// TwinCAT 3 PLC project SaftyPLC_1
// ProgramVersion: 3.1.4026.12
// libraries:
//   Tc2_Standard, * (Beckhoff Automation GmbH)
//   Tc2_System, * (Beckhoff Automation GmbH)
//   Tc2_Utilities, * (Beckhoff Automation GmbH)
//   Tc3_Module, * (Beckhoff Automation GmbH)
// project tree:
//   GVLs/ GVL_io.TcGVL, GVL_Safety.TcGVL
//   / PlcTask.TcTTO, XTS_Task.TcTTO (not stored)
//   POUs/ MAIN.TcPOU
// (motion and I/O tree: see PLC project planartrackmovement_1)
// real-time tasks:
//   TASK XTS Task: cycle T#500us, priority 1, ADS port 350
//   TASK Job Task: cycle default, priority 32
//   TASK MC-Task (MET): cycle T#2ms, priority 3, ADS port 521
//   TASK MC-Task (MPT): cycle T#10ms, priority 8, ADS port 531
//   TASK PlcTask: cycle T#1ms, priority 20, ADS port 351
//   TASK PlcTask1: cycle T#1ms, priority 21, ADS port 352
// variable links:
//   SaftyPLC_1/SaftyPLC_1 Instance <-> Device 1 (EtherCAT)/Term 1 (EK1200)/Term 13 (EL2912)
//     PlcTask Inputs/GVL_Safety.Error_Com <-> StandardInputs/TwinSafeGroup1.Error_Com_142
//     PlcTask Inputs/GVL_Safety.Error_Other <-> StandardInputs/TwinSafeGroup1.Error_Other_143
//     PlcTask Inputs/GVL_Safety.Error_Out <-> StandardInputs/TwinSafeGroup1.Error_out_141
//     PlcTask Inputs/GVL_Safety.SaeftyOk <-> StandardInputs/TwinSafeGroup1.SafetyOk_72
//     PlcTask Inputs/GVL_Safety.SafetyInRun <-> StandardInputs/TwinSafeGroup1.SafetyInRun_73
//     PlcTask Outputs/GVL_Safety.Reset <-> StandardOutputs/TwinSafeGroup1.ErrorAcknowledgement_1
//     PlcTask Outputs/GVL_Safety.Run <-> StandardOutputs/TwinSafeGroup1.Run_2
//     PlcTask Outputs/GVL_Safety.Start <-> StandardOutputs/TwinSafeGroup1.STO_75
//   SaftyPLC_1/SaftyPLC_1 Instance <-> Device 1 (EtherCAT)/Term 1 (EK1200)/Term 2 (EL1809)
//     PlcTask Inputs/GVL_Safety.HwReset <-> Channel 16/Input
//     PlcTask Inputs/GVL_Safety.HwStart <-> Channel 14/Input
//     PlcTask Inputs/GVL_Safety.HwStop <-> Channel 15/Input
//   SaftyPLC_1/SaftyPLC_1 Instance <-> Device 4 (EtherCAT)/Box 50 (AT5100-0100)
//     PlcTask Inputs/GVL_io.D_Spannung[5] <-> DRV Info data 1/D-Spannung
//     PlcTask Inputs/GVL_io.Q_Spannung[5] <-> DRV Info data 1/Q-Spannung
//     PlcTask Outputs/GVL_Safety.Reset <-> Module 1 (SAFETY)/SAFETY Standard Outputdata/Standard In Var 1
//     PlcTask Outputs/GVL_Safety.Run <-> Module 1 (SAFETY)/SAFETY Standard Outputdata/Standard In Var 5
//   SaftyPLC_1/SaftyPLC_1 Instance <-> Device 4 (EtherCAT)/Box 51 (AT5100-0100)
//     PlcTask Inputs/GVL_io.D_Spannung[6] <-> DRV Info data 1/D-Spannung
//     PlcTask Inputs/GVL_io.Q_Spannung[6] <-> DRV Info data 1/Q-Spannung
//     PlcTask Outputs/GVL_Safety.Reset <-> Module 1 (SAFETY)/SAFETY Standard Outputdata/Standard In Var 1
//     PlcTask Outputs/GVL_Safety.Run <-> Module 1 (SAFETY)/SAFETY Standard Outputdata/Standard In Var 5
//   SaftyPLC_1/SaftyPLC_1 Instance <-> Device 4 (EtherCAT)/Box 52 (AT5100-0100)
//     PlcTask Outputs/GVL_Safety.Reset <-> Module 1 (SAFETY)/SAFETY Standard Outputdata/Standard In Var 1
//     PlcTask Outputs/GVL_Safety.Run <-> Module 1 (SAFETY)/SAFETY Standard Outputdata/Standard In Var 5
//   SaftyPLC_1/SaftyPLC_1 Instance <-> Device 4 (EtherCAT)/Box 53 (AT5100-0100)
//     PlcTask Outputs/GVL_Safety.Reset <-> Module 1 (SAFETY)/SAFETY Standard Outputdata/Standard In Var 1
//     PlcTask Outputs/GVL_Safety.Run <-> Module 1 (SAFETY)/SAFETY Standard Outputdata/Standard In Var 5
//   SaftyPLC_1/SaftyPLC_1 Instance <-> Device 4 (EtherCAT)/Box 54 (AT5100-0100)
//     PlcTask Outputs/GVL_Safety.Reset <-> Module 1 (SAFETY)/SAFETY Standard Outputdata/Standard In Var 1
//     PlcTask Outputs/GVL_Safety.Run <-> Module 1 (SAFETY)/SAFETY Standard Outputdata/Standard In Var 5
//   SaftyPLC_1/SaftyPLC_1 Instance <-> Device 4 (EtherCAT)/Box 55 (AT5100-0100)
//     PlcTask Outputs/GVL_Safety.Reset <-> Module 1 (SAFETY)/SAFETY Standard Outputdata/Standard In Var 1
//     PlcTask Outputs/GVL_Safety.Run <-> Module 1 (SAFETY)/SAFETY Standard Outputdata/Standard In Var 5
//   SaftyPLC_1/SaftyPLC_1 Instance <-> Device 4 (EtherCAT)/Box 56 (AT5100-0100)
//     PlcTask Outputs/GVL_Safety.Reset <-> Module 1 (SAFETY)/SAFETY Standard Outputdata/Standard In Var 1
//     PlcTask Outputs/GVL_Safety.Run <-> Module 1 (SAFETY)/SAFETY Standard Outputdata/Standard In Var 5
//   SaftyPLC_1/SaftyPLC_1 Instance <-> Device 4 (EtherCAT)/Box 57 (AT5100-0100)
//     PlcTask Outputs/GVL_Safety.Reset <-> Module 1 (SAFETY)/SAFETY Standard Outputdata/Standard In Var 1
//     PlcTask Outputs/GVL_Safety.Run <-> Module 1 (SAFETY)/SAFETY Standard Outputdata/Standard In Var 5
//   SaftyPLC_1/SaftyPLC_1 Instance <-> Device 4 (EtherCAT)/Box 58 (AT5100-0100)
//     PlcTask Outputs/GVL_Safety.Reset <-> Module 1 (SAFETY)/SAFETY Standard Outputdata/Standard In Var 1
//     PlcTask Outputs/GVL_Safety.Run <-> Module 1 (SAFETY)/SAFETY Standard Outputdata/Standard In Var 5
//   SaftyPLC_1/SaftyPLC_1 Instance <-> Device 4 (EtherCAT)/Box 59 (AT5100-0100)
//     PlcTask Outputs/GVL_Safety.Reset <-> Module 1 (SAFETY)/SAFETY Standard Outputdata/Standard In Var 1
//     PlcTask Outputs/GVL_Safety.Run <-> Module 1 (SAFETY)/SAFETY Standard Outputdata/Standard In Var 5
//   SaftyPLC_1/SaftyPLC_1 Instance <-> Device 4 (EtherCAT)/Box 60 (AT5100-0100)
//     PlcTask Outputs/GVL_Safety.Reset <-> Module 1 (SAFETY)/SAFETY Standard Outputdata/Standard In Var 1
//     PlcTask Outputs/GVL_Safety.Run <-> Module 1 (SAFETY)/SAFETY Standard Outputdata/Standard In Var 5
//   SaftyPLC_1/SaftyPLC_1 Instance <-> Device 4 (EtherCAT)/Box 61 (AT5100-0100)
//     PlcTask Outputs/GVL_Safety.Reset <-> Module 1 (SAFETY)/SAFETY Standard Outputdata/Standard In Var 1
//     PlcTask Outputs/GVL_Safety.Run <-> Module 1 (SAFETY)/SAFETY Standard Outputdata/Standard In Var 5
//   SaftyPLC_1/SaftyPLC_1 Instance <-> Device 4 (EtherCAT)/Box 62 (AT5100-0100)
//     PlcTask Outputs/GVL_Safety.Reset <-> Module 1 (SAFETY)/SAFETY Standard Outputdata/Standard In Var 1
//     PlcTask Outputs/GVL_Safety.Run <-> Module 1 (SAFETY)/SAFETY Standard Outputdata/Standard In Var 5
//   SaftyPLC_1/SaftyPLC_1 Instance <-> Device 4 (EtherCAT)/Box 63 (AT5100-0100)
//     PlcTask Outputs/GVL_Safety.Reset <-> Module 1 (SAFETY)/SAFETY Standard Outputdata/Standard In Var 1
//     PlcTask Outputs/GVL_Safety.Run <-> Module 1 (SAFETY)/SAFETY Standard Outputdata/Standard In Var 5
//   SaftyPLC_1/SaftyPLC_1 Instance <-> Device 4 (EtherCAT)/Box 64 (AT5100-0100)
//     PlcTask Outputs/GVL_Safety.Reset <-> Module 1 (SAFETY)/SAFETY Standard Outputdata/Standard In Var 1
//     PlcTask Outputs/GVL_Safety.Run <-> Module 1 (SAFETY)/SAFETY Standard Outputdata/Standard In Var 5
//   SaftyPLC_1/SaftyPLC_1 Instance <-> Device 4 (EtherCAT)/Box 65 (AT5100-0100)
//     PlcTask Outputs/GVL_Safety.Reset <-> Module 1 (SAFETY)/SAFETY Standard Outputdata/Standard In Var 1
//     PlcTask Outputs/GVL_Safety.Run <-> Module 1 (SAFETY)/SAFETY Standard Outputdata/Standard In Var 5
//   SaftyPLC_1/SaftyPLC_1 Instance <-> Device 4 (EtherCAT)/Box 66 (AT5100-0100)
//     PlcTask Outputs/GVL_Safety.Reset <-> Module 1 (SAFETY)/SAFETY Standard Outputdata/Standard In Var 1
//     PlcTask Outputs/GVL_Safety.Run <-> Module 1 (SAFETY)/SAFETY Standard Outputdata/Standard In Var 5
//   SaftyPLC_1/SaftyPLC_1 Instance <-> Device 4 (EtherCAT)/Box 67 (AT5100-0100)
//     PlcTask Outputs/GVL_Safety.Reset <-> Module 1 (SAFETY)/SAFETY Standard Outputdata/Standard In Var 1
//     PlcTask Outputs/GVL_Safety.Run <-> Module 1 (SAFETY)/SAFETY Standard Outputdata/Standard In Var 5
//   SaftyPLC_1/SaftyPLC_1 Instance <-> Device 4 (EtherCAT)/Box 68 (AT5100-0100)
//     PlcTask Outputs/GVL_Safety.Reset <-> Module 1 (SAFETY)/SAFETY Standard Outputdata/Standard In Var 1
//     PlcTask Outputs/GVL_Safety.Run <-> Module 1 (SAFETY)/SAFETY Standard Outputdata/Standard In Var 5
//   SaftyPLC_1/SaftyPLC_1 Instance <-> Device 4 (EtherCAT)/Box 69 (AT5100-0100)
//     PlcTask Outputs/GVL_Safety.Reset <-> Module 1 (SAFETY)/SAFETY Standard Outputdata/Standard In Var 1
//     PlcTask Outputs/GVL_Safety.Run <-> Module 1 (SAFETY)/SAFETY Standard Outputdata/Standard In Var 5
//   SaftyPLC_1/SaftyPLC_1 Instance <-> Device 4 (EtherCAT)/Box 70 (AT5100-0100)
//     PlcTask Outputs/GVL_Safety.Reset <-> Module 1 (SAFETY)/SAFETY Standard Outputdata/Standard In Var 1
//     PlcTask Outputs/GVL_Safety.Run <-> Module 1 (SAFETY)/SAFETY Standard Outputdata/Standard In Var 5
//   SaftyPLC_1/SaftyPLC_1 Instance <-> Device 4 (EtherCAT)/Box 71 (AT5100-0100)
//     PlcTask Outputs/GVL_Safety.Reset <-> Module 1 (SAFETY)/SAFETY Standard Outputdata/Standard In Var 1
//     PlcTask Outputs/GVL_Safety.Run <-> Module 1 (SAFETY)/SAFETY Standard Outputdata/Standard In Var 5
//   SaftyPLC_1/SaftyPLC_1 Instance <-> Device 4 (EtherCAT)/Box 72 (AT5100-0100)
//     PlcTask Outputs/GVL_Safety.Reset <-> Module 1 (SAFETY)/SAFETY Standard Outputdata/Standard In Var 1
//     PlcTask Outputs/GVL_Safety.Run <-> Module 1 (SAFETY)/SAFETY Standard Outputdata/Standard In Var 5
//   SaftyPLC_1/SaftyPLC_1 Instance <-> Device 4 (EtherCAT)/Box 73 (AT5100-0100)
//     PlcTask Outputs/GVL_Safety.Reset <-> Module 1 (SAFETY)/SAFETY Standard Outputdata/Standard In Var 1
//     PlcTask Outputs/GVL_Safety.Run <-> Module 1 (SAFETY)/SAFETY Standard Outputdata/Standard In Var 5
//   SaftyPLC_1/SaftyPLC_1 Instance <-> Device 4 (EtherCAT)/Box 74 (AT5100-0100)
//     PlcTask Outputs/GVL_Safety.Reset <-> Module 1 (SAFETY)/SAFETY Standard Outputdata/Standard In Var 1
//     PlcTask Outputs/GVL_Safety.Run <-> Module 1 (SAFETY)/SAFETY Standard Outputdata/Standard In Var 5
//   SaftyPLC_1/SaftyPLC_1 Instance <-> Device 4 (EtherCAT)/Box 75 (AT5100-0100)
//     PlcTask Outputs/GVL_Safety.Reset <-> Module 1 (SAFETY)/SAFETY Standard Outputdata/Standard In Var 1
//     PlcTask Outputs/GVL_Safety.Run <-> Module 1 (SAFETY)/SAFETY Standard Outputdata/Standard In Var 5
//   SaftyPLC_1/SaftyPLC_1 Instance <-> Device 4 (EtherCAT)/Box 76 (AT5100-0100)
//     PlcTask Outputs/GVL_Safety.Reset <-> Module 1 (SAFETY)/SAFETY Standard Outputdata/Standard In Var 1
//     PlcTask Outputs/GVL_Safety.Run <-> Module 1 (SAFETY)/SAFETY Standard Outputdata/Standard In Var 5
//   SaftyPLC_1/SaftyPLC_1 Instance <-> Device 4 (EtherCAT)/Box 77 (AT5100-0100)
//     PlcTask Outputs/GVL_Safety.Reset <-> Module 1 (SAFETY)/SAFETY Standard Outputdata/Standard In Var 1
//     PlcTask Outputs/GVL_Safety.Run <-> Module 1 (SAFETY)/SAFETY Standard Outputdata/Standard In Var 5
//   SaftyPLC_1/SaftyPLC_1 Instance <-> Device 4 (EtherCAT)/Box 78 (AT5100-0100)
//     PlcTask Outputs/GVL_Safety.Reset <-> Module 1 (SAFETY)/SAFETY Standard Outputdata/Standard In Var 1
//     PlcTask Outputs/GVL_Safety.Run <-> Module 1 (SAFETY)/SAFETY Standard Outputdata/Standard In Var 5
//   SaftyPLC_1/SaftyPLC_1 Instance <-> Device 4 (EtherCAT)/Box 79 (AT5100-0100)
//     PlcTask Outputs/GVL_Safety.Reset <-> Module 1 (SAFETY)/SAFETY Standard Outputdata/Standard In Var 1
//     PlcTask Outputs/GVL_Safety.Run <-> Module 1 (SAFETY)/SAFETY Standard Outputdata/Standard In Var 5
//   SaftyPLC_1/SaftyPLC_1 Instance <-> Device 4 (EtherCAT)/Box 80 (AT5100-0100)
//     PlcTask Inputs/GVL_io.D_Spannung[7] <-> DRV Info data 1/D-Spannung
//     PlcTask Inputs/GVL_io.Q_Spannung[7] <-> DRV Info data 1/Q-Spannung
//     PlcTask Outputs/GVL_Safety.Reset <-> Module 1 (SAFETY)/SAFETY Standard Outputdata/Standard In Var 1
//     PlcTask Outputs/GVL_Safety.Run <-> Module 1 (SAFETY)/SAFETY Standard Outputdata/Standard In Var 5
//   SaftyPLC_1/SaftyPLC_1 Instance <-> Device 4 (EtherCAT)/Box 81 (AT5100-0100)
//     PlcTask Inputs/GVL_io.D_Spannung[8] <-> DRV Info data 1/D-Spannung
//     PlcTask Inputs/GVL_io.Q_Spannung[8] <-> DRV Info data 1/Q-Spannung
//     PlcTask Outputs/GVL_Safety.Reset <-> Module 1 (SAFETY)/SAFETY Standard Outputdata/Standard In Var 1
//     PlcTask Outputs/GVL_Safety.Run <-> Module 1 (SAFETY)/SAFETY Standard Outputdata/Standard In Var 5
//   SaftyPLC_1/SaftyPLC_1 Instance <-> Device 8 (EtherCAT)/Box 18 (AT5100-0100)
//     PlcTask Inputs/GVL_io.D_Spannung[1] <-> DRV Info data 1/D-Spannung
//     PlcTask Inputs/GVL_io.Q_Spannung[1] <-> DRV Info data 1/Q-Spannung
//     PlcTask Outputs/GVL_Safety.Reset <-> Module 1 (SAFETY)/SAFETY Standard Outputdata/Standard In Var 1
//     PlcTask Outputs/GVL_Safety.Run <-> Module 1 (SAFETY)/SAFETY Standard Outputdata/Standard In Var 5
//   SaftyPLC_1/SaftyPLC_1 Instance <-> Device 8 (EtherCAT)/Box 19 (AT5100-0100)
//     PlcTask Inputs/GVL_io.D_Spannung[2] <-> DRV Info data 1/D-Spannung
//     PlcTask Inputs/GVL_io.Q_Spannung[2] <-> DRV Info data 1/Q-Spannung
//     PlcTask Outputs/GVL_Safety.Reset <-> Module 1 (SAFETY)/SAFETY Standard Outputdata/Standard In Var 1
//     PlcTask Outputs/GVL_Safety.Run <-> Module 1 (SAFETY)/SAFETY Standard Outputdata/Standard In Var 5
//   SaftyPLC_1/SaftyPLC_1 Instance <-> Device 8 (EtherCAT)/Box 20 (AT5100-0100)
//     PlcTask Outputs/GVL_Safety.Reset <-> Module 1 (SAFETY)/SAFETY Standard Outputdata/Standard In Var 1
//     PlcTask Outputs/GVL_Safety.Run <-> Module 1 (SAFETY)/SAFETY Standard Outputdata/Standard In Var 5
//   SaftyPLC_1/SaftyPLC_1 Instance <-> Device 8 (EtherCAT)/Box 21 (AT5100-0100)
//     PlcTask Outputs/GVL_Safety.Reset <-> Module 1 (SAFETY)/SAFETY Standard Outputdata/Standard In Var 1
//     PlcTask Outputs/GVL_Safety.Run <-> Module 1 (SAFETY)/SAFETY Standard Outputdata/Standard In Var 5
//   SaftyPLC_1/SaftyPLC_1 Instance <-> Device 8 (EtherCAT)/Box 22 (AT5100-0100)
//     PlcTask Outputs/GVL_Safety.Reset <-> Module 1 (SAFETY)/SAFETY Standard Outputdata/Standard In Var 1
//     PlcTask Outputs/GVL_Safety.Run <-> Module 1 (SAFETY)/SAFETY Standard Outputdata/Standard In Var 5
//   SaftyPLC_1/SaftyPLC_1 Instance <-> Device 8 (EtherCAT)/Box 23 (AT5100-0100)
//     PlcTask Outputs/GVL_Safety.Reset <-> Module 1 (SAFETY)/SAFETY Standard Outputdata/Standard In Var 1
//     PlcTask Outputs/GVL_Safety.Run <-> Module 1 (SAFETY)/SAFETY Standard Outputdata/Standard In Var 5
//   SaftyPLC_1/SaftyPLC_1 Instance <-> Device 8 (EtherCAT)/Box 24 (AT5100-0100)
//     PlcTask Outputs/GVL_Safety.Reset <-> Module 1 (SAFETY)/SAFETY Standard Outputdata/Standard In Var 1
//     PlcTask Outputs/GVL_Safety.Run <-> Module 1 (SAFETY)/SAFETY Standard Outputdata/Standard In Var 5
//   SaftyPLC_1/SaftyPLC_1 Instance <-> Device 8 (EtherCAT)/Box 25 (AT5100-0100)
//     PlcTask Outputs/GVL_Safety.Reset <-> Module 1 (SAFETY)/SAFETY Standard Outputdata/Standard In Var 1
//     PlcTask Outputs/GVL_Safety.Run <-> Module 1 (SAFETY)/SAFETY Standard Outputdata/Standard In Var 5
//   SaftyPLC_1/SaftyPLC_1 Instance <-> Device 8 (EtherCAT)/Box 26 (AT5100-0100)
//     PlcTask Outputs/GVL_Safety.Reset <-> Module 1 (SAFETY)/SAFETY Standard Outputdata/Standard In Var 1
//     PlcTask Outputs/GVL_Safety.Run <-> Module 1 (SAFETY)/SAFETY Standard Outputdata/Standard In Var 5
//   SaftyPLC_1/SaftyPLC_1 Instance <-> Device 8 (EtherCAT)/Box 27 (AT5100-0100)
//     PlcTask Outputs/GVL_Safety.Reset <-> Module 1 (SAFETY)/SAFETY Standard Outputdata/Standard In Var 1
//     PlcTask Outputs/GVL_Safety.Run <-> Module 1 (SAFETY)/SAFETY Standard Outputdata/Standard In Var 5
//   SaftyPLC_1/SaftyPLC_1 Instance <-> Device 8 (EtherCAT)/Box 28 (AT5100-0100)
//     PlcTask Outputs/GVL_Safety.Reset <-> Module 1 (SAFETY)/SAFETY Standard Outputdata/Standard In Var 1
//     PlcTask Outputs/GVL_Safety.Run <-> Module 1 (SAFETY)/SAFETY Standard Outputdata/Standard In Var 5
//   SaftyPLC_1/SaftyPLC_1 Instance <-> Device 8 (EtherCAT)/Box 29 (AT5100-0100)
//     PlcTask Outputs/GVL_Safety.Reset <-> Module 1 (SAFETY)/SAFETY Standard Outputdata/Standard In Var 1
//     PlcTask Outputs/GVL_Safety.Run <-> Module 1 (SAFETY)/SAFETY Standard Outputdata/Standard In Var 5
//   SaftyPLC_1/SaftyPLC_1 Instance <-> Device 8 (EtherCAT)/Box 30 (AT5100-0100)
//     PlcTask Outputs/GVL_Safety.Reset <-> Module 1 (SAFETY)/SAFETY Standard Outputdata/Standard In Var 1
//     PlcTask Outputs/GVL_Safety.Run <-> Module 1 (SAFETY)/SAFETY Standard Outputdata/Standard In Var 5
//   SaftyPLC_1/SaftyPLC_1 Instance <-> Device 8 (EtherCAT)/Box 31 (AT5100-0100)
//     PlcTask Outputs/GVL_Safety.Reset <-> Module 1 (SAFETY)/SAFETY Standard Outputdata/Standard In Var 1
//     PlcTask Outputs/GVL_Safety.Run <-> Module 1 (SAFETY)/SAFETY Standard Outputdata/Standard In Var 5
//   SaftyPLC_1/SaftyPLC_1 Instance <-> Device 8 (EtherCAT)/Box 32 (AT5100-0100)
//     PlcTask Outputs/GVL_Safety.Reset <-> Module 1 (SAFETY)/SAFETY Standard Outputdata/Standard In Var 1
//     PlcTask Outputs/GVL_Safety.Run <-> Module 1 (SAFETY)/SAFETY Standard Outputdata/Standard In Var 5
//   SaftyPLC_1/SaftyPLC_1 Instance <-> Device 8 (EtherCAT)/Box 33 (AT5100-0100)
//     PlcTask Outputs/GVL_Safety.Reset <-> Module 1 (SAFETY)/SAFETY Standard Outputdata/Standard In Var 1
//     PlcTask Outputs/GVL_Safety.Run <-> Module 1 (SAFETY)/SAFETY Standard Outputdata/Standard In Var 5
//   SaftyPLC_1/SaftyPLC_1 Instance <-> Device 8 (EtherCAT)/Box 34 (AT5100-0100)
//     PlcTask Outputs/GVL_Safety.Reset <-> Module 1 (SAFETY)/SAFETY Standard Outputdata/Standard In Var 1
//     PlcTask Outputs/GVL_Safety.Run <-> Module 1 (SAFETY)/SAFETY Standard Outputdata/Standard In Var 5
//   SaftyPLC_1/SaftyPLC_1 Instance <-> Device 8 (EtherCAT)/Box 35 (AT5100-0100)
//     PlcTask Outputs/GVL_Safety.Reset <-> Module 1 (SAFETY)/SAFETY Standard Outputdata/Standard In Var 1
//     PlcTask Outputs/GVL_Safety.Run <-> Module 1 (SAFETY)/SAFETY Standard Outputdata/Standard In Var 5
//   SaftyPLC_1/SaftyPLC_1 Instance <-> Device 8 (EtherCAT)/Box 36 (AT5100-0100)
//     PlcTask Outputs/GVL_Safety.Reset <-> Module 1 (SAFETY)/SAFETY Standard Outputdata/Standard In Var 1
//     PlcTask Outputs/GVL_Safety.Run <-> Module 1 (SAFETY)/SAFETY Standard Outputdata/Standard In Var 5
//   SaftyPLC_1/SaftyPLC_1 Instance <-> Device 8 (EtherCAT)/Box 37 (AT5100-0100)
//     PlcTask Outputs/GVL_Safety.Reset <-> Module 1 (SAFETY)/SAFETY Standard Outputdata/Standard In Var 1
//     PlcTask Outputs/GVL_Safety.Run <-> Module 1 (SAFETY)/SAFETY Standard Outputdata/Standard In Var 5
//   SaftyPLC_1/SaftyPLC_1 Instance <-> Device 8 (EtherCAT)/Box 38 (AT5100-0100)
//     PlcTask Outputs/GVL_Safety.Reset <-> Module 1 (SAFETY)/SAFETY Standard Outputdata/Standard In Var 1
//     PlcTask Outputs/GVL_Safety.Run <-> Module 1 (SAFETY)/SAFETY Standard Outputdata/Standard In Var 5
//   SaftyPLC_1/SaftyPLC_1 Instance <-> Device 8 (EtherCAT)/Box 39 (AT5100-0100)
//     PlcTask Outputs/GVL_Safety.Reset <-> Module 1 (SAFETY)/SAFETY Standard Outputdata/Standard In Var 1
//     PlcTask Outputs/GVL_Safety.Run <-> Module 1 (SAFETY)/SAFETY Standard Outputdata/Standard In Var 5
//   SaftyPLC_1/SaftyPLC_1 Instance <-> Device 8 (EtherCAT)/Box 40 (AT5100-0100)
//     PlcTask Outputs/GVL_Safety.Reset <-> Module 1 (SAFETY)/SAFETY Standard Outputdata/Standard In Var 1
//     PlcTask Outputs/GVL_Safety.Run <-> Module 1 (SAFETY)/SAFETY Standard Outputdata/Standard In Var 5
//   SaftyPLC_1/SaftyPLC_1 Instance <-> Device 8 (EtherCAT)/Box 41 (AT5100-0100)
//     PlcTask Outputs/GVL_Safety.Reset <-> Module 1 (SAFETY)/SAFETY Standard Outputdata/Standard In Var 1
//     PlcTask Outputs/GVL_Safety.Run <-> Module 1 (SAFETY)/SAFETY Standard Outputdata/Standard In Var 5
//   SaftyPLC_1/SaftyPLC_1 Instance <-> Device 8 (EtherCAT)/Box 42 (AT5100-0100)
//     PlcTask Outputs/GVL_Safety.Reset <-> Module 1 (SAFETY)/SAFETY Standard Outputdata/Standard In Var 1
//     PlcTask Outputs/GVL_Safety.Run <-> Module 1 (SAFETY)/SAFETY Standard Outputdata/Standard In Var 5
//   SaftyPLC_1/SaftyPLC_1 Instance <-> Device 8 (EtherCAT)/Box 43 (AT5100-0100)
//     PlcTask Outputs/GVL_Safety.Reset <-> Module 1 (SAFETY)/SAFETY Standard Outputdata/Standard In Var 1
//     PlcTask Outputs/GVL_Safety.Run <-> Module 1 (SAFETY)/SAFETY Standard Outputdata/Standard In Var 5
//   SaftyPLC_1/SaftyPLC_1 Instance <-> Device 8 (EtherCAT)/Box 44 (AT5100-0100)
//     PlcTask Outputs/GVL_Safety.Reset <-> Module 1 (SAFETY)/SAFETY Standard Outputdata/Standard In Var 1
//     PlcTask Outputs/GVL_Safety.Run <-> Module 1 (SAFETY)/SAFETY Standard Outputdata/Standard In Var 5
//   SaftyPLC_1/SaftyPLC_1 Instance <-> Device 8 (EtherCAT)/Box 45 (AT5100-0100)
//     PlcTask Outputs/GVL_Safety.Reset <-> Module 1 (SAFETY)/SAFETY Standard Outputdata/Standard In Var 1
//     PlcTask Outputs/GVL_Safety.Run <-> Module 1 (SAFETY)/SAFETY Standard Outputdata/Standard In Var 5
//   SaftyPLC_1/SaftyPLC_1 Instance <-> Device 8 (EtherCAT)/Box 46 (AT5100-0100)
//     PlcTask Outputs/GVL_Safety.Reset <-> Module 1 (SAFETY)/SAFETY Standard Outputdata/Standard In Var 1
//     PlcTask Outputs/GVL_Safety.Run <-> Module 1 (SAFETY)/SAFETY Standard Outputdata/Standard In Var 5
//   SaftyPLC_1/SaftyPLC_1 Instance <-> Device 8 (EtherCAT)/Box 47 (AT5100-0100)
//     PlcTask Outputs/GVL_Safety.Reset <-> Module 1 (SAFETY)/SAFETY Standard Outputdata/Standard In Var 1
//     PlcTask Outputs/GVL_Safety.Run <-> Module 1 (SAFETY)/SAFETY Standard Outputdata/Standard In Var 5
//   SaftyPLC_1/SaftyPLC_1 Instance <-> Device 8 (EtherCAT)/Box 48 (AT5100-0100)
//     PlcTask Inputs/GVL_io.D_Spannung[3] <-> DRV Info data 1/D-Spannung
//     PlcTask Inputs/GVL_io.Q_Spannung[3] <-> DRV Info data 1/Q-Spannung
//     PlcTask Outputs/GVL_Safety.Reset <-> Module 1 (SAFETY)/SAFETY Standard Outputdata/Standard In Var 1
//     PlcTask Outputs/GVL_Safety.Run <-> Module 1 (SAFETY)/SAFETY Standard Outputdata/Standard In Var 5
//   SaftyPLC_1/SaftyPLC_1 Instance <-> Device 8 (EtherCAT)/Box 49 (AT5100-0100)
//     PlcTask Inputs/GVL_io.D_Spannung[4] <-> DRV Info data 1/D-Spannung
//     PlcTask Inputs/GVL_io.Q_Spannung[4] <-> DRV Info data 1/Q-Spannung
//     PlcTask Outputs/GVL_Safety.Reset <-> Module 1 (SAFETY)/SAFETY Standard Outputdata/Standard In Var 1
//     PlcTask Outputs/GVL_Safety.Run <-> Module 1 (SAFETY)/SAFETY Standard Outputdata/Standard In Var 5

CONFIGURATION SaftyPLC_1
    RESOURCE PLC ON TwinCAT3
        TASK PlcTask(INTERVAL := T#1ms, PRIORITY := 20);
        PROGRAM MAIN WITH PlcTask : MAIN;
    END_RESOURCE
END_CONFIGURATION

// ---- GVLs/GVL_io.TcGVL

VAR_GLOBAL
	Q_Spannung AT%I*: ARRAY[1..10] OF REAL;
	D_Spannung AT%I*: ARRAY[1..10] OF REAL;
	Voltage : ARRAY[1..10] OF REAL; 
END_VAR

// ---- GVLs/GVL_Safety.TcGVL
{attribute 'qualified_only'}
VAR_GLOBAL
	Run			AT%Q* : BOOL := TRUE;
	Start		AT%Q* : BOOL := TRUE;
	Reset		AT%Q* : BOOL;
	
	SafetyInRun	AT%I* : BOOL;
	SaeftyOk 	AT%I* : BOOL;
	
	Error_Other	AT%I* : BOOL;
	Error_Out	AT%I* : BOOL;
	Error_Com	AT%I* : BOOL;
	
	HwStart 	AT%I* : BOOL;
	HwStop		AT%I* : BOOL;
	HwReset 	AT%I* : BOOL;
	
	HW_Ok			AT%Q* : BOOL;
	HW_Error	 	AT%Q* : BOOL;
	HW_Reset_Req 	AT%Q* : BOOL;
 
END_VAR

// ---- POUs/MAIN.TcPOU
PROGRAM MAIN
VAR
	nState,i: INT;
	fbR_TrigExecute : R_Trig;
	StartSafety :BOOL := TRUE;
	
	TcRestart : TC_Restart;
	Restart : BOOL;
	busy : BOOL;
	State AT%I* :ARRAY[1..2] OF UINT;
END_VAR

FOR i := 1 TO 8 DO 
	GVL_io.Voltage[i]:= SQRT( EXP(GVL_io.D_Spannung[i]) + EXP(GVL_io.Q_Spannung[i]));
END_FOR


IF GVL_Safety.hwStart THEN
	StartSafety := TRUE;
	GVL_Safety.Run := TRUE;
	GVL_Safety.Start := TRUE;

ELSIF NOT GVL_Safety.hwStop	THEN 
	StartSafety := FALSE;
END_IF

GVL_Safety.Reset := GVL_Safety.hwReset  OR Restart;

 GVL_Safety.HW_Error :=  State[1] <> 8 OR  State[2] <> 8  ;
GVL_Safety.HW_Ok  :=GVL_Safety.SaeftyOk;

 GVL_Safety.HW_Reset_Req:= (GVL_Safety.Error_Other OR GVL_Safety.Error_Out OR GVL_Safety.Error_Com );
(*
TcRestart(
	NETID:= '', 
	RESTART:=Restart , 
	TMOUT:= , 
	BUSY=> busy, 
	ERR=> , 
	ERRID=> );
	
	*)

METHOD Safety : BOOL

VAR_INPUT
	bExecute : BOOL;
END_VAR

VAR

END_VAR
fbR_TrigExecute(CLK := bExecute);
IF fbR_TrigExecute.Q   THEN
	nState := 10;		
ELSIF NOT bExecute THEN
	nState := 0;
	GVL_Safety.Run := FALSE;
	
END_IF

CASE nState OF
	 0: // Wait State
	 	
	10: 
		GVL_Safety.Run := TRUE;
		GVL_Safety.Start := TRUE;
		GVL_Safety.Reset := TRUE;
		nState :=20;
	15:

		GVL_Safety.Reset := FALSE;
		nState :=200;

			
	20:
		GVL_Safety.Reset := FALSE;

		IF 	GVL_Safety.SaeftyOk THEN
			nState :=99;
			Safety := TRUE;
		ELSIF 	(GVL_Safety.Error_Other OR GVL_Safety.Error_Out OR GVL_Safety.Error_Com )  THEN 
		
			nState :=15;
		END_IF
	40:
		GVL_Safety.reset := TRUE;
		IF NOT (GVL_Safety.Error_Other OR GVL_Safety.Error_Out OR GVL_Safety.Error_Com )THEN
			GVL_Safety.Reset := FALSE;
			nState :=99;
		END_IF	
	99: 
		IF NOT GVL_Safety.SaeftyOk THEN
			nState :=40;
			Safety := TRUE;
		END_IF

	
END_CASE
END_METHOD

END_PROGRAM
